{attribute addProperty BoxType "EL3632-0000-0022"}
{attribute addProperty Id "Sample_CountAT %I*UINT162"}
{attribute addProperty CRC "1190388509"}
{attribute addProperty SizeInBites "16"}
{attribute addProperty SizeInBytes "2"}
TYPE Sample_Count_46F3E31D :
STRUCT
	{attribute addProperty Name "Sample_Count"}
	Sample_Count AT %I* : UINT;
END_STRUCT
END_TYPE

(* stored: Version 1.2.0.0, ProductVersion 3.1.4024.9
   DUT Sample_Count_46F3E31D: Id {c674f8ba-1988-4604-80d5-5d529bde756d} *)
